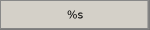
VISUALIZATION HMI_Button  // 150x30
VAR_INPUT
	i_sText : STRING;
END_VAR
VAR_IN_OUT
	iq_stButton : ST_HmiButton;
END_VAR
    Button (0,0 150x30), "%s", text variable: i_sText, pressed state: iq_stButton.stToHmi.bProcessState, invisible if: iq_stButton.stToHmi.bInvisible, input disabled if: not iq_stButton.stToHmi.bEnabled
        tap iq_stButton.stFromHmi.bPressed
END_VISUALIZATION

(* stored: Version 1.1.0.1, ProductVersion 3.1.4026.13
   Visu HMI_Button: Id {3d10b32c-8d65-49ea-bc1a-47c9b2c0a658} *)
